// SIMATIC STEP 7 (V5.x) project evaluacion1
// CPU: CPU317-2
// station: Hardware
// station: SIMATIC 300(1)
// station: P_ADR_BUS
// program: S7 Program(1)

SYMBOL_TABLE
"Ejercicio1"	FB 1	FB 1
"Ejercicio 2"	FB 2	FB 2
"Ejercicio3"	FB 3	FB 3
"Ejercicio 4"	FB 4	FB 4
"Ejercicio 5"	FB 5	FB 5
"Ejercicio 6"	FB 6	FB 6
"Ejercicio C1"	FB 7	FB 7
"Ejercicio C2"	FB 8	FB 8
"Ejercicio 3-5"	FB 9	FB 9
"Ejercicio 3-6"	FB 10	FB 10
"Ejercicio 3-7"	FB 11	FB 11
"Ejercicio 6-1"	FB 12	FB 12
"Ejercicio 6-2"	FB 13	FB 13
"Ejercicio 6-3"	FB 14	FB 14
"Paro de emergencia"	FB 99	FB 99
"CYCL_EXC"	OB 1	OB 1	// Cycle Execution
END_SYMBOL_TABLE

FUNCTION_BLOCK "Ejercicio1"	// FB 1
TITLE = Ejercicio 1
VERSION : 0.1
VAR_INPUT
  C_CONTINUO : BOOL ;
  C_UNICO : BOOL ;
  PARO : BOOL ;
  DET_PIEZA : BOOL ;
  A0 : BOOL ;
  A1 : BOOL ;
  B0 : BOOL ;
  B1 : BOOL ;
  C0 : BOOL ;
  C1 : BOOL ;
END_VAR
VAR_OUTPUT
  Y1 : BOOL ;
  Y2 : BOOL ;
  Y3 : BOOL ;
  Y4 : BOOL ;
  Y5 : BOOL ;
  Y6 : BOOL ;
END_VAR
VAR
  K_UNI : BOOL ;
  K_CON : BOOL ;
  K0 : BOOL ;
  K1 : BOOL ;
  K2 : BOOL ;
  K3 : BOOL ;
  K4 : BOOL ;
  K5 : BOOL ;
  K6 : BOOL ;
END_VAR
BEGIN
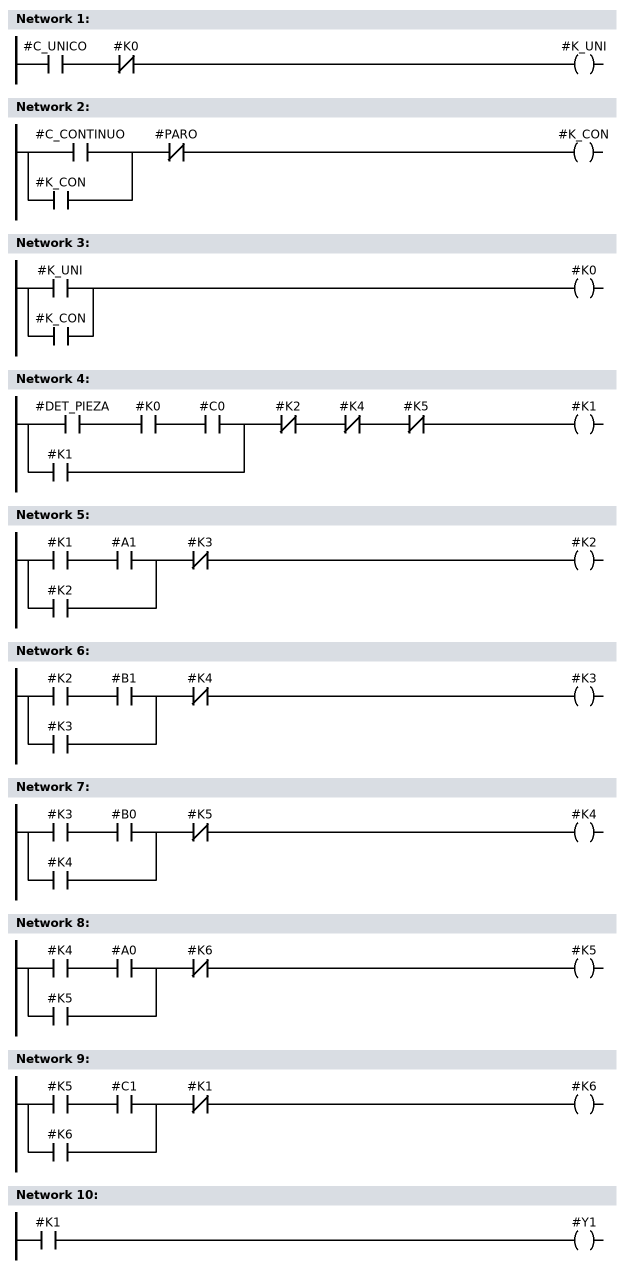
NETWORK
TITLE =
      A     #C_UNICO;
      AN    #K0;
      =     #K_UNI;
NETWORK
TITLE =
      A(;
      O     #C_CONTINUO;
      O     #K_CON;
      );
      AN    #PARO;
      =     #K_CON;
NETWORK
TITLE =
      O     #K_UNI;
      O     #K_CON;
      =     #K0;
NETWORK
TITLE =
      A(;
      A     #DET_PIEZA;
      A     #K0;
      A     #C0;
      O     #K1;
      );
      AN    #K2;
      AN    #K4;
      AN    #K5;
      =     #K1;
NETWORK
TITLE =
      A(;
      A     #K1;
      A     #A1;
      O     #K2;
      );
      AN    #K3;
      =     #K2;
NETWORK
TITLE =
      A(;
      A     #K2;
      A     #B1;
      O     #K3;
      );
      AN    #K4;
      =     #K3;
NETWORK
TITLE =
      A(;
      A     #K3;
      A     #B0;
      O     #K4;
      );
      AN    #K5;
      =     #K4;
NETWORK
TITLE =
      A(;
      A     #K4;
      A     #A0;
      O     #K5;
      );
      AN    #K6;
      =     #K5;
NETWORK
TITLE =
      A(;
      A     #K5;
      A     #C1;
      O     #K6;
      );
      AN    #K1;
      =     #K6;
NETWORK
TITLE =
      A     #K1;
      =     #Y1;
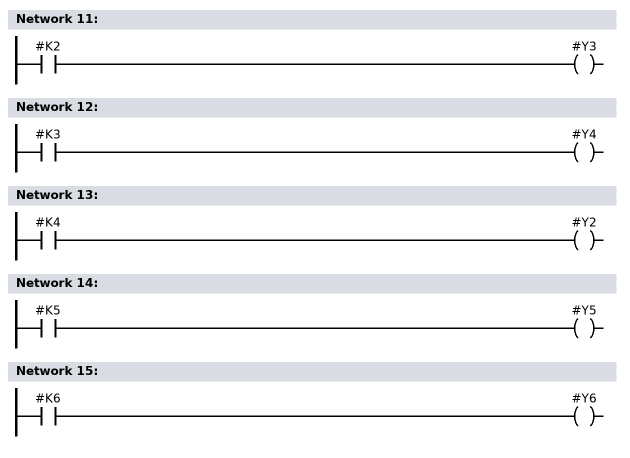
NETWORK
TITLE =
      A     #K2;
      =     #Y3;
NETWORK
TITLE =
      A     #K3;
      =     #Y4;
NETWORK
TITLE =
      A     #K4;
      =     #Y2;
NETWORK
TITLE =
      A     #K5;
      =     #Y5;
NETWORK
TITLE =
      A     #K6;
      =     #Y6;
END_FUNCTION_BLOCK

FUNCTION_BLOCK "Ejercicio 2"	// FB 2
TITLE = Ejercicio 2
VERSION : 0.1
VAR_INPUT
  C_UNICO : BOOL ;
  A0 : BOOL ;
  A1 : BOOL ;
  B0 : BOOL ;
  B1 : BOOL ;
  C0 : BOOL ;
  C1 : BOOL ;
END_VAR
VAR_OUTPUT
  Y1 : BOOL ;
  Y2 : BOOL ;
  Y3 : BOOL ;
  Y4 : BOOL ;
  Y5 : BOOL ;
  Y6 : BOOL ;
END_VAR
VAR
  K_UNI : BOOL ;
  K0 : BOOL ;
  K1 : BOOL ;
  K2 : BOOL ;
  K3 : BOOL ;
  K4 : BOOL ;
  K5 : BOOL ;
  K6 : BOOL ;
END_VAR
BEGIN
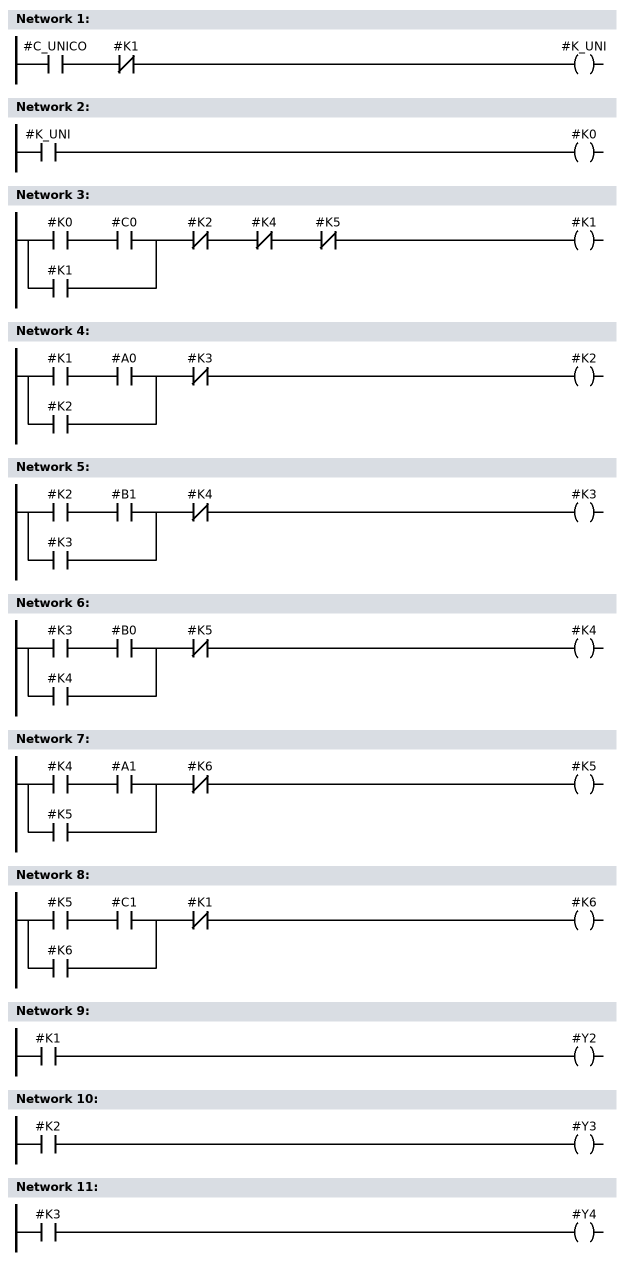
NETWORK
TITLE =
      A     #C_UNICO;
      AN    #K1;
      =     #K_UNI;
NETWORK
TITLE =
      A     #K_UNI;
      =     #K0;
NETWORK
TITLE =
      A(;
      A     #K0;
      A     #C0;
      O     #K1;
      );
      AN    #K2;
      AN    #K4;
      AN    #K5;
      =     #K1;
NETWORK
TITLE =
      A(;
      A     #K1;
      A     #A0;
      O     #K2;
      );
      AN    #K3;
      =     #K2;
NETWORK
TITLE =
      A(;
      A     #K2;
      A     #B1;
      O     #K3;
      );
      AN    #K4;
      =     #K3;
NETWORK
TITLE =
      A(;
      A     #K3;
      A     #B0;
      O     #K4;
      );
      AN    #K5;
      =     #K4;
NETWORK
TITLE =
      A(;
      A     #K4;
      A     #A1;
      O     #K5;
      );
      AN    #K6;
      =     #K5;
NETWORK
TITLE =
      A(;
      A     #K5;
      A     #C1;
      O     #K6;
      );
      AN    #K1;
      =     #K6;
NETWORK
TITLE =
      A     #K1;
      =     #Y2;
NETWORK
TITLE =
      A     #K2;
      =     #Y3;
NETWORK
TITLE =
      A     #K3;
      =     #Y4;
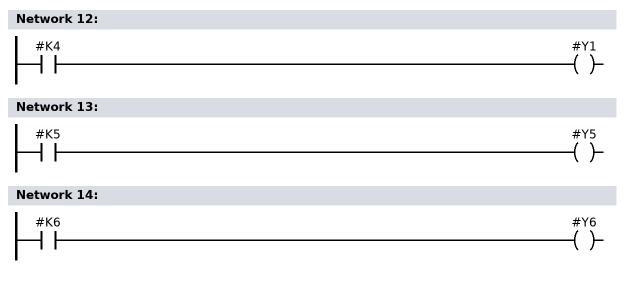
NETWORK
TITLE =
      A     #K4;
      =     #Y1;
NETWORK
TITLE =
      A     #K5;
      =     #Y5;
NETWORK
TITLE =
      A     #K6;
      =     #Y6;
END_FUNCTION_BLOCK

FUNCTION_BLOCK "Ejercicio3"	// FB 3
VERSION : 0.1
VAR_INPUT
  C_UNICO : BOOL ;
  A0 : BOOL ;
  A1 : BOOL ;
  B0 : BOOL ;
  B1 : BOOL ;
  C0 : BOOL ;
  C1 : BOOL ;
END_VAR
VAR_OUTPUT
  Y1 : BOOL ;
  Y2 : BOOL ;
  Y3 : BOOL ;
  Y4 : BOOL ;
  Y5 : BOOL ;
  Y6 : BOOL ;
END_VAR
VAR
  K0 : BOOL ;
  K1 : BOOL ;
  K2 : BOOL ;
  K3 : BOOL ;
  K4 : BOOL ;
  K5 : BOOL ;
  K6 : BOOL ;
  K_UNI : BOOL ;
END_VAR
BEGIN
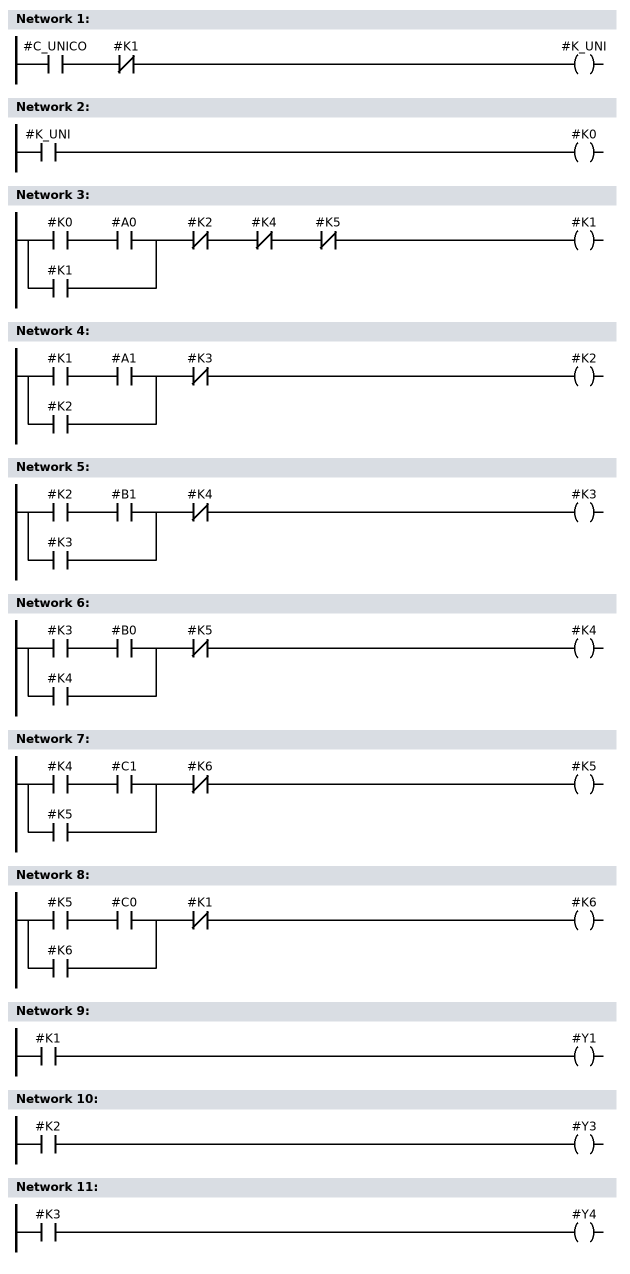
NETWORK
TITLE =
      A     #C_UNICO;
      AN    #K1;
      =     #K_UNI;
NETWORK
TITLE =
      A     #K_UNI;
      =     #K0;
NETWORK
TITLE =
      A(;
      A     #K0;
      A     #A0;
      O     #K1;
      );
      AN    #K2;
      AN    #K4;
      AN    #K5;
      =     #K1;
NETWORK
TITLE =
      A(;
      A     #K1;
      A     #A1;
      O     #K2;
      );
      AN    #K3;
      =     #K2;
NETWORK
TITLE =
      A(;
      A     #K2;
      A     #B1;
      O     #K3;
      );
      AN    #K4;
      =     #K3;
NETWORK
TITLE =
      A(;
      A     #K3;
      A     #B0;
      O     #K4;
      );
      AN    #K5;
      =     #K4;
NETWORK
TITLE =
      A(;
      A     #K4;
      A     #C1;
      O     #K5;
      );
      AN    #K6;
      =     #K5;
NETWORK
TITLE =
      A(;
      A     #K5;
      A     #C0;
      O     #K6;
      );
      AN    #K1;
      =     #K6;
NETWORK
TITLE =
      A     #K1;
      =     #Y1;
NETWORK
TITLE =
      A     #K2;
      =     #Y3;
NETWORK
TITLE =
      A     #K3;
      =     #Y4;
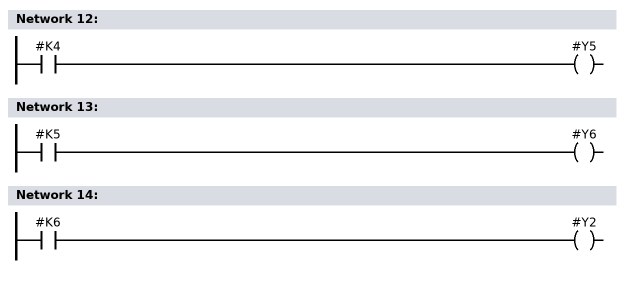
NETWORK
TITLE =
      A     #K4;
      =     #Y5;
NETWORK
TITLE =
      A     #K5;
      =     #Y6;
NETWORK
TITLE =
      A     #K6;
      =     #Y2;
END_FUNCTION_BLOCK

FUNCTION_BLOCK "Ejercicio 4"	// FB 4
VERSION : 0.1
VAR_INPUT
  C_UNICO : BOOL ;
  C_CONTINUO : BOOL ;
  A0 : BOOL ;
  A1 : BOOL ;
  B0 : BOOL ;
  B1 : BOOL ;
  C0 : BOOL ;
  C1 : BOOL ;
  D0 : BOOL ;
  D1 : BOOL ;
  PARO : BOOL ;
END_VAR
VAR_OUTPUT
  Y1 : BOOL ;
  Y2 : BOOL ;
  Y3 : BOOL ;
  Y4 : BOOL ;
  Y5 : BOOL ;
  Y6 : BOOL ;
  Y7 : BOOL ;
  Y8 : BOOL ;
END_VAR
VAR
  K_UNI : BOOL ;
  K_CON : BOOL ;
  K0 : BOOL ;
  K1 : BOOL ;
  K2 : BOOL ;
  K3 : BOOL ;
  K4 : BOOL ;
  K5 : BOOL ;
  K6 : BOOL ;
  K7 : BOOL ;
  K8 : BOOL ;
END_VAR
BEGIN
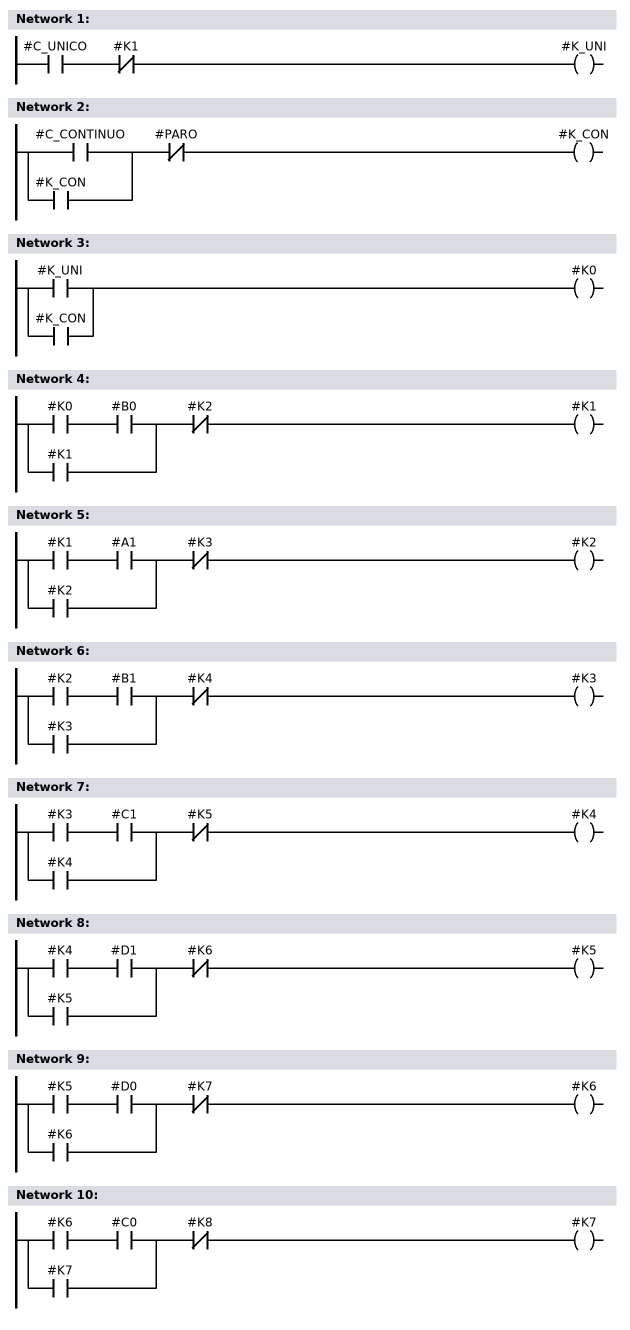
NETWORK
TITLE =
      A     #C_UNICO;
      AN    #K1;
      =     #K_UNI;
NETWORK
TITLE =
      A(;
      O     #C_CONTINUO;
      O     #K_CON;
      );
      AN    #PARO;
      =     #K_CON;
NETWORK
TITLE =
      O     #K_UNI;
      O     #K_CON;
      =     #K0;
NETWORK
TITLE =
      A(;
      A     #K0;
      A     #B0;
      O     #K1;
      );
      AN    #K2;
      =     #K1;
NETWORK
TITLE =
      A(;
      A     #K1;
      A     #A1;
      O     #K2;
      );
      AN    #K3;
      =     #K2;
NETWORK
TITLE =
      A(;
      A     #K2;
      A     #B1;
      O     #K3;
      );
      AN    #K4;
      =     #K3;
NETWORK
TITLE =
      A(;
      A     #K3;
      A     #C1;
      O     #K4;
      );
      AN    #K5;
      =     #K4;
NETWORK
TITLE =
      A(;
      A     #K4;
      A     #D1;
      O     #K5;
      );
      AN    #K6;
      =     #K5;
NETWORK
TITLE =
      A(;
      A     #K5;
      A     #D0;
      O     #K6;
      );
      AN    #K7;
      =     #K6;
NETWORK
TITLE =
      A(;
      A     #K6;
      A     #C0;
      O     #K7;
      );
      AN    #K8;
      =     #K7;
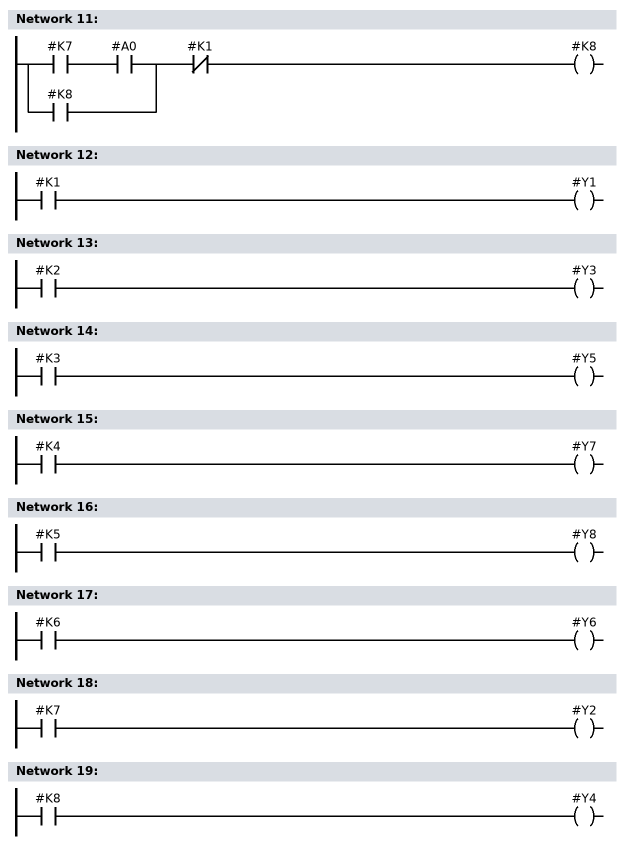
NETWORK
TITLE =
      A(;
      A     #K7;
      A     #A0;
      O     #K8;
      );
      AN    #K1;
      =     #K8;
NETWORK
TITLE =
      A     #K1;
      =     #Y1;
NETWORK
TITLE =
      A     #K2;
      =     #Y3;
NETWORK
TITLE =
      A     #K3;
      =     #Y5;
NETWORK
TITLE =
      A     #K4;
      =     #Y7;
NETWORK
TITLE =
      A     #K5;
      =     #Y8;
NETWORK
TITLE =
      A     #K6;
      =     #Y6;
NETWORK
TITLE =
      A     #K7;
      =     #Y2;
NETWORK
TITLE =
      A     #K8;
      =     #Y4;
END_FUNCTION_BLOCK

FUNCTION_BLOCK "Ejercicio 5"	// FB 5
VERSION : 0.1
VAR_INPUT
  C_UNICO : BOOL ;
  A0 : BOOL ;
  A1 : BOOL ;
  B0 : BOOL ;
  B1 : BOOL ;
  C0 : BOOL ;
  C1 : BOOL ;
END_VAR
VAR_OUTPUT
  Y1 : BOOL ;
  Y2 : BOOL ;
  Y3 : BOOL ;
  Y4 : BOOL ;
  Y5 : BOOL ;
  Y6 : BOOL ;
END_VAR
VAR
  K_UNI : BOOL ;
  K0 : BOOL ;
  K1 : BOOL ;
  K2 : BOOL ;
  K3 : BOOL ;
  K4 : BOOL ;
  K5 : BOOL ;
  K6 : BOOL ;
  K7 : BOOL ;
  K8 : BOOL ;
  K9 : BOOL ;
  K10 : BOOL ;
END_VAR
BEGIN
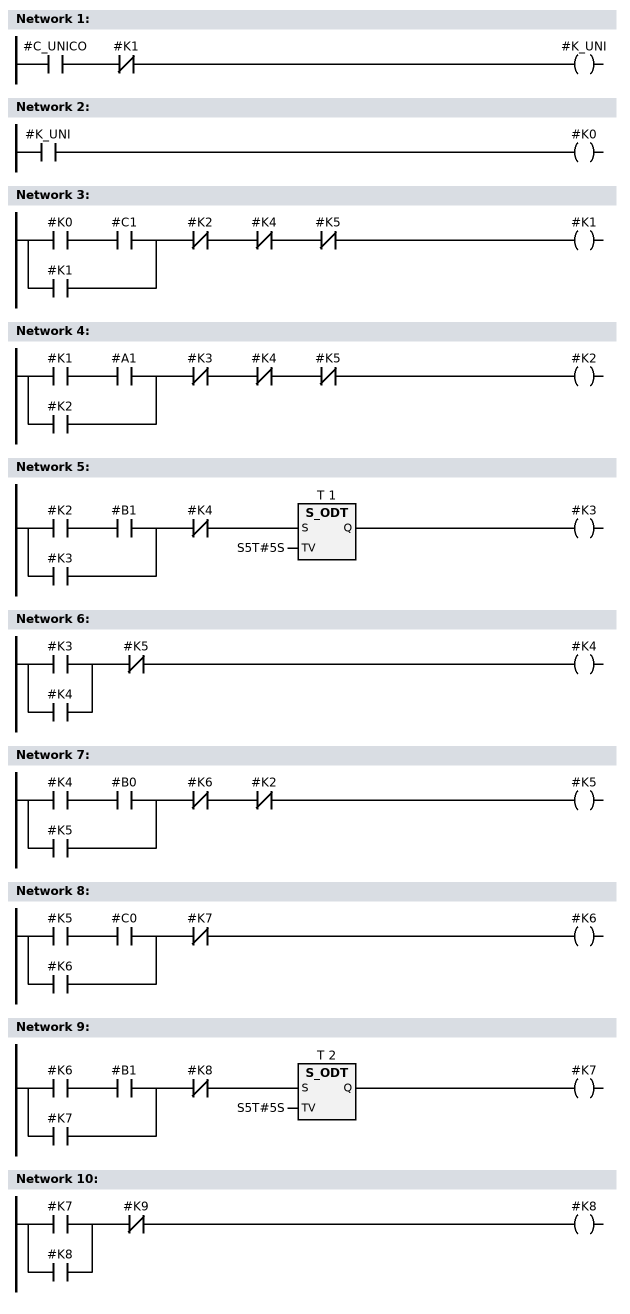
NETWORK
TITLE =
      A     #C_UNICO;
      AN    #K1;
      =     #K_UNI;
NETWORK
TITLE =
      A     #K_UNI;
      =     #K0;
NETWORK
TITLE =
      A(;
      A     #K0;
      A     #C1;
      O     #K1;
      );
      AN    #K2;
      AN    #K4;
      AN    #K5;
      =     #K1;
NETWORK
TITLE =
      A(;
      A     #K1;
      A     #A1;
      O     #K2;
      );
      AN    #K3;
      AN    #K4;
      AN    #K5;
      =     #K2;
NETWORK
TITLE =
      A(;
      A     #K2;
      A     #B1;
      O     #K3;
      );
      AN    #K4;
      L     S5T#5S;
      SD    T 1;
      NOP   0;
      NOP   0;
      NOP   0;
      A     T 1;
      =     #K3;
NETWORK
TITLE =
      A(;
      O     #K3;
      O     #K4;
      );
      AN    #K5;
      =     #K4;
NETWORK
TITLE =
      A(;
      A     #K4;
      A     #B0;
      O     #K5;
      );
      AN    #K6;
      AN    #K2;
      =     #K5;
NETWORK
TITLE =
      A(;
      A     #K5;
      A     #C0;
      O     #K6;
      );
      AN    #K7;
      =     #K6;
NETWORK
TITLE =
      A(;
      A     #K6;
      A     #B1;
      O     #K7;
      );
      AN    #K8;
      L     S5T#5S;
      SD    T 2;
      NOP   0;
      NOP   0;
      NOP   0;
      A     T 2;
      =     #K7;
NETWORK
TITLE =
      A(;
      O     #K7;
      O     #K8;
      );
      AN    #K9;
      =     #K8;
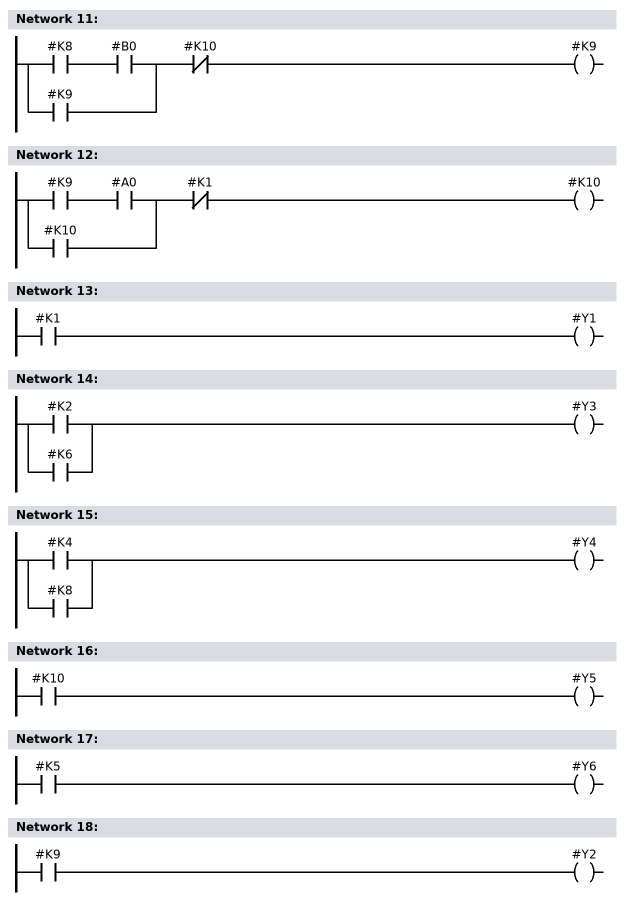
NETWORK
TITLE =
      A(;
      A     #K8;
      A     #B0;
      O     #K9;
      );
      AN    #K10;
      =     #K9;
NETWORK
TITLE =
      A(;
      A     #K9;
      A     #A0;
      O     #K10;
      );
      AN    #K1;
      =     #K10;
NETWORK
TITLE =
      A     #K1;
      =     #Y1;
NETWORK
TITLE =
      O     #K2;
      O     #K6;
      =     #Y3;
NETWORK
TITLE =
      O     #K4;
      O     #K8;
      =     #Y4;
NETWORK
TITLE =
      A     #K10;
      =     #Y5;
NETWORK
TITLE =
      A     #K5;
      =     #Y6;
NETWORK
TITLE =
      A     #K9;
      =     #Y2;
END_FUNCTION_BLOCK

FUNCTION_BLOCK "Ejercicio 6"	// FB 6
VERSION : 0.1
VAR_INPUT
  C_UNICO : BOOL ;
  C_CONTINUO : BOOL ;
  PARO : BOOL ;
  A0 : BOOL ;
  A1 : BOOL ;
  B0 : BOOL ;
  B1 : BOOL ;
  C0 : BOOL ;
  C1 : BOOL ;
  D0 : BOOL ;
  D1 : BOOL ;
END_VAR
VAR_OUTPUT
  Y1 : BOOL ;
  Y2 : BOOL ;
  Y3 : BOOL ;
  Y4 : BOOL ;
  Y5 : BOOL ;
  Y6 : BOOL ;
  Y7 : BOOL ;
  Y8 : BOOL ;
END_VAR
VAR
  K0 : BOOL ;
  K1 : BOOL ;
  K2 : BOOL ;
  K3 : BOOL ;
  K4 : BOOL ;
  K5 : BOOL ;
  K6 : BOOL ;
  K7 : BOOL ;
  K8 : BOOL ;
  KA : BOOL ;
  KB : BOOL ;
END_VAR
BEGIN
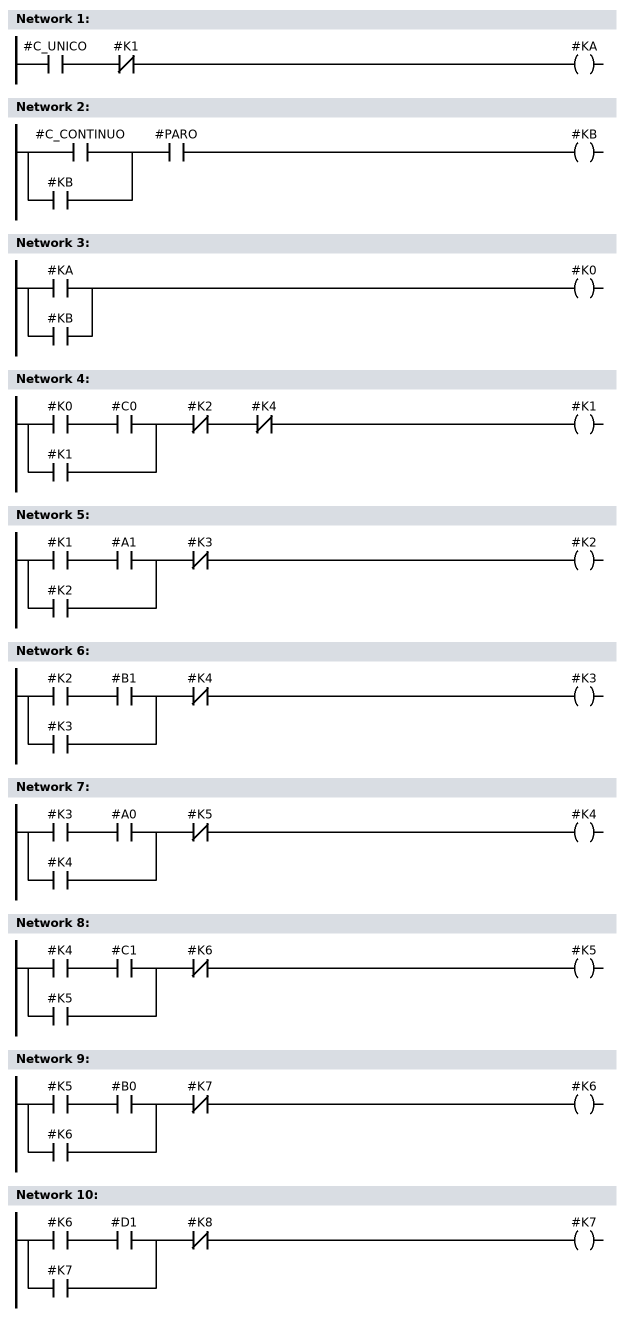
NETWORK
TITLE =
      A     #C_UNICO;
      AN    #K1;
      =     #KA;
NETWORK
TITLE =
      A(;
      O     #C_CONTINUO;
      O     #KB;
      );
      A     #PARO;
      =     #KB;
NETWORK
TITLE =
      O     #KA;
      O     #KB;
      =     #K0;
NETWORK
TITLE =
      A(;
      A     #K0;
      A     #C0;
      O     #K1;
      );
      AN    #K2;
      AN    #K4;
      =     #K1;
NETWORK
TITLE =
      A(;
      A     #K1;
      A     #A1;
      O     #K2;
      );
      AN    #K3;
      =     #K2;
NETWORK
TITLE =
      A(;
      A     #K2;
      A     #B1;
      O     #K3;
      );
      AN    #K4;
      =     #K3;
NETWORK
TITLE =
      A(;
      A     #K3;
      A     #A0;
      O     #K4;
      );
      AN    #K5;
      =     #K4;
NETWORK
TITLE =
      A(;
      A     #K4;
      A     #C1;
      O     #K5;
      );
      AN    #K6;
      =     #K5;
NETWORK
TITLE =
      A(;
      A     #K5;
      A     #B0;
      O     #K6;
      );
      AN    #K7;
      =     #K6;
NETWORK
TITLE =
      A(;
      A     #K6;
      A     #D1;
      O     #K7;
      );
      AN    #K8;
      =     #K7;
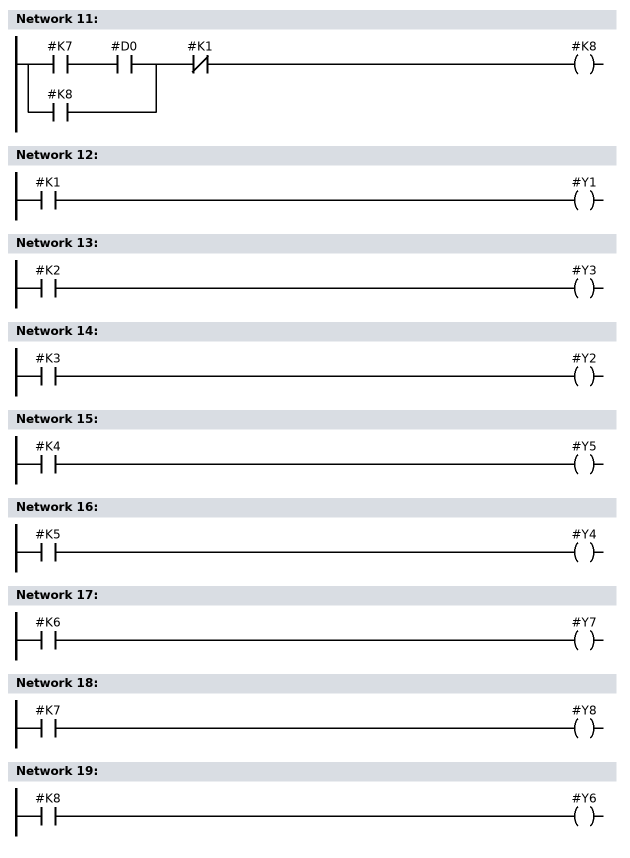
NETWORK
TITLE =
      A(;
      A     #K7;
      A     #D0;
      O     #K8;
      );
      AN    #K1;
      =     #K8;
NETWORK
TITLE =
      A     #K1;
      =     #Y1;
NETWORK
TITLE =
      A     #K2;
      =     #Y3;
NETWORK
TITLE =
      A     #K3;
      =     #Y2;
NETWORK
TITLE =
      A     #K4;
      =     #Y5;
NETWORK
TITLE =
      A     #K5;
      =     #Y4;
NETWORK
TITLE =
      A     #K6;
      =     #Y7;
NETWORK
TITLE =
      A     #K7;
      =     #Y8;
NETWORK
TITLE =
      A     #K8;
      =     #Y6;
END_FUNCTION_BLOCK

FUNCTION_BLOCK "Ejercicio C1"	// FB 7
VERSION : 0.1
VAR_INPUT
  C_UNICO : BOOL ;
  C_CONTINUO : BOOL ;
  PARO : BOOL ;
  C_BROCA : BOOL ;
  A0 : BOOL ;
  A1 : BOOL ;
  B0 : BOOL ;
  B1 : BOOL ;
  C0 : BOOL ;
  C1 : BOOL ;
END_VAR
VAR_OUTPUT
  Y1 : BOOL ;
  Y2 : BOOL ;
  Y3 : BOOL ;
  Y4 : BOOL ;
  Y5 : BOOL ;
  Y6 : BOOL ;
END_VAR
VAR
  K0 : BOOL ;
  K1 : BOOL ;
  K2 : BOOL ;
  K3 : BOOL ;
  K4 : BOOL ;
  K5 : BOOL ;
  K6 : BOOL ;
  KA : BOOL ;
  KB : BOOL ;
  CNT : BOOL ;
  K7 : BOOL ;
  K8 : BOOL ;
  K9 : BOOL ;
  K10 : BOOL ;
  K11 : BOOL ;
  K12 : BOOL ;
END_VAR
BEGIN
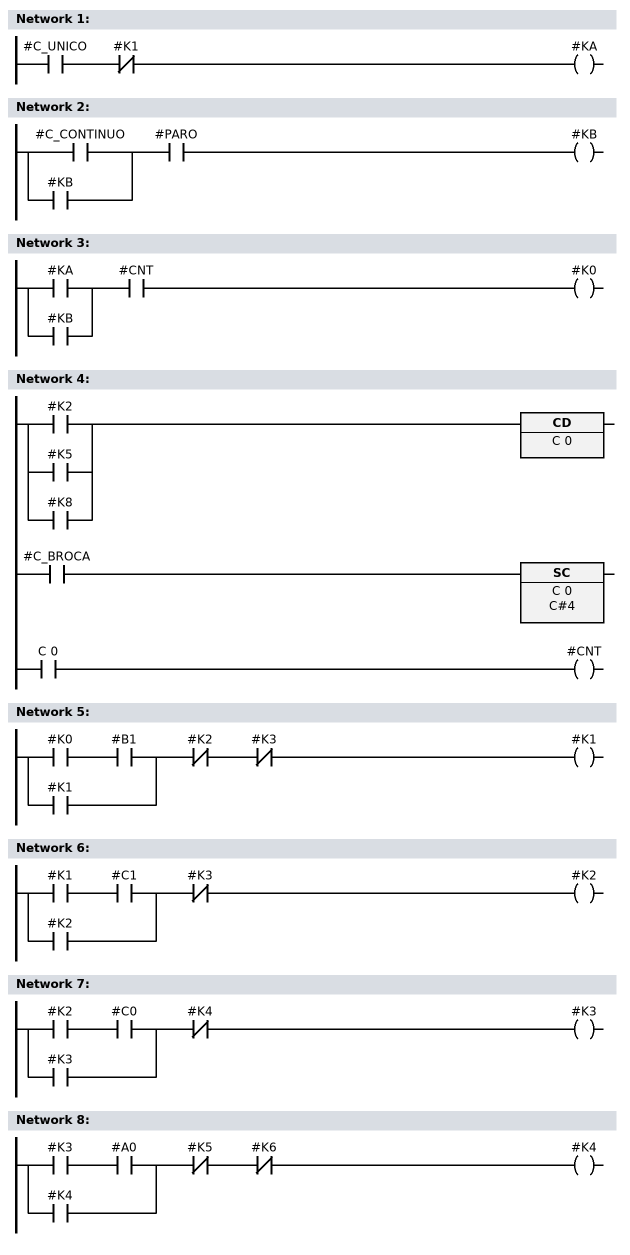
NETWORK
TITLE =
      A     #C_UNICO;
      AN    #K1;
      =     #KA;
NETWORK
TITLE =
      A(;
      O     #C_CONTINUO;
      O     #KB;
      );
      A     #PARO;
      =     #KB;
NETWORK
TITLE =
      A(;
      O     #KA;
      O     #KB;
      );
      A     #CNT;
      =     #K0;
NETWORK
TITLE =
      A(;
      O     #K2;
      O     #K5;
      O     #K8;
      );
      CD    C 0;
      BLD   101;
      A     #C_BROCA;
      L     C#4;
      S     C 0;
      NOP   0;
      NOP   0;
      NOP   0;
      A     C 0;
      =     #CNT;
NETWORK
TITLE =
      A(;
      A     #K0;
      A     #B1;
      O     #K1;
      );
      AN    #K2;
      AN    #K3;
      =     #K1;
NETWORK
TITLE =
      A(;
      A     #K1;
      A     #C1;
      O     #K2;
      );
      AN    #K3;
      =     #K2;
NETWORK
TITLE =
      A(;
      A     #K2;
      A     #C0;
      O     #K3;
      );
      AN    #K4;
      =     #K3;
NETWORK
TITLE =
      A(;
      A     #K3;
      A     #A0;
      O     #K4;
      );
      AN    #K5;
      AN    #K6;
      =     #K4;
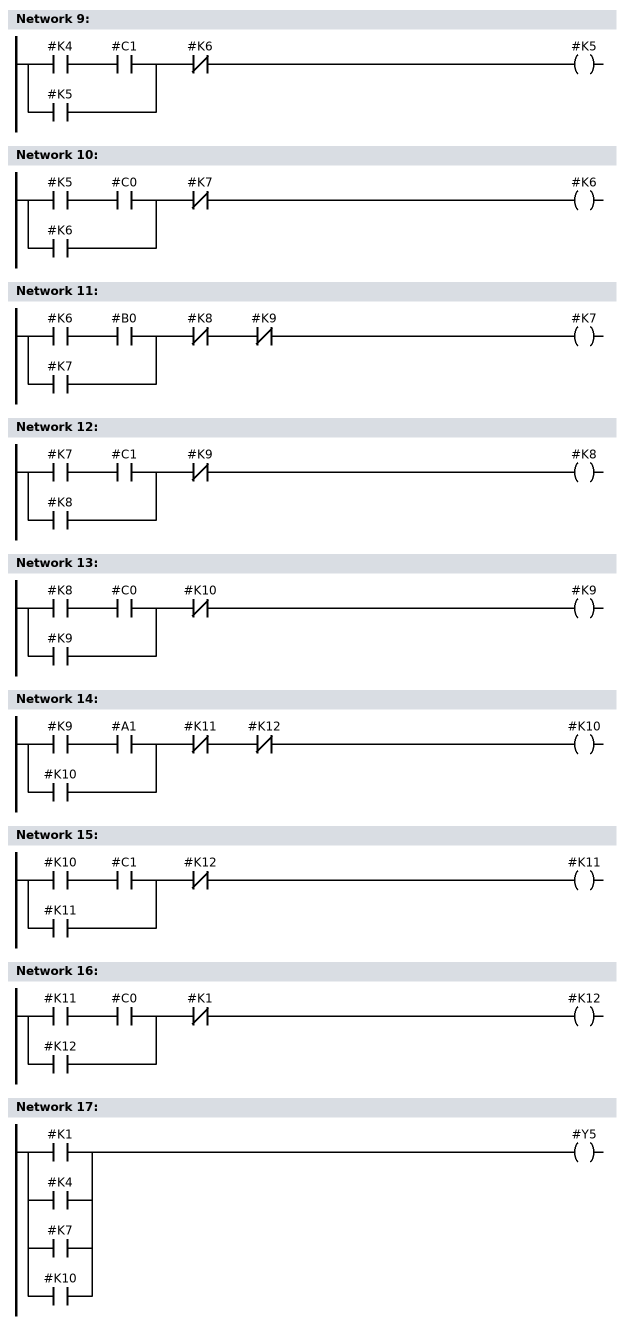
NETWORK
TITLE =
      A(;
      A     #K4;
      A     #C1;
      O     #K5;
      );
      AN    #K6;
      =     #K5;
NETWORK
TITLE =
      A(;
      A     #K5;
      A     #C0;
      O     #K6;
      );
      AN    #K7;
      =     #K6;
NETWORK
TITLE =
      A(;
      A     #K6;
      A     #B0;
      O     #K7;
      );
      AN    #K8;
      AN    #K9;
      =     #K7;
NETWORK
TITLE =
      A(;
      A     #K7;
      A     #C1;
      O     #K8;
      );
      AN    #K9;
      =     #K8;
NETWORK
TITLE =
      A(;
      A     #K8;
      A     #C0;
      O     #K9;
      );
      AN    #K10;
      =     #K9;
NETWORK
TITLE =
      A(;
      A     #K9;
      A     #A1;
      O     #K10;
      );
      AN    #K11;
      AN    #K12;
      =     #K10;
NETWORK
TITLE =
      A(;
      A     #K10;
      A     #C1;
      O     #K11;
      );
      AN    #K12;
      =     #K11;
NETWORK
TITLE =
      A(;
      A     #K11;
      A     #C0;
      O     #K12;
      );
      AN    #K1;
      =     #K12;
NETWORK
TITLE =
      O     #K1;
      O     #K4;
      O     #K7;
      O     #K10;
      =     #Y5;
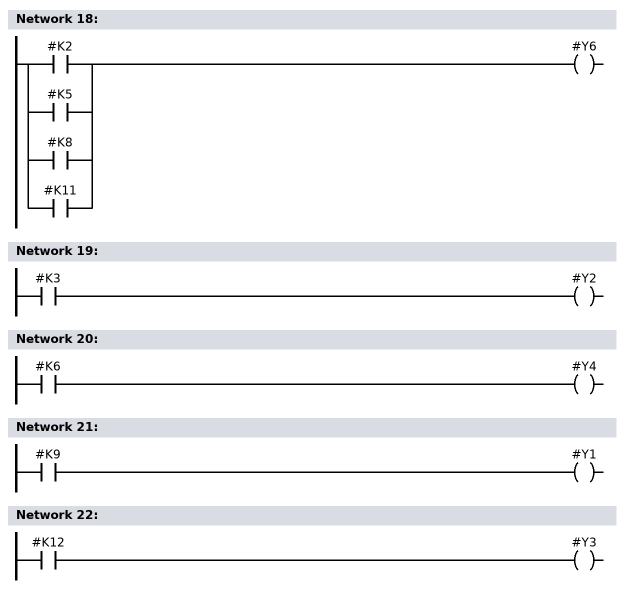
NETWORK
TITLE =
      O     #K2;
      O     #K5;
      O     #K8;
      O     #K11;
      =     #Y6;
NETWORK
TITLE =
      A     #K3;
      =     #Y2;
NETWORK
TITLE =
      A     #K6;
      =     #Y4;
NETWORK
TITLE =
      A     #K9;
      =     #Y1;
NETWORK
TITLE =
      A     #K12;
      =     #Y3;
END_FUNCTION_BLOCK

FUNCTION_BLOCK "Ejercicio C2"	// FB 8
VERSION : 0.1
VAR_INPUT
  C_UNICO : BOOL ;
  C_CONTINUO : BOOL ;
  PARO : BOOL ;
  DET_PIEZA : BOOL ;
  DET_CINTA : BOOL ;
  A0 : BOOL ;
  A1 : BOOL ;
  B0 : BOOL ;
  B1 : BOOL ;
  C0 : BOOL ;
  C1 : BOOL ;
  D0 : BOOL ;
  D1 : BOOL ;
  E0 : BOOL ;
  E1 : BOOL ;
  F0 : BOOL ;
  F1 : BOOL ;
END_VAR
VAR_OUTPUT
  Y1 : BOOL ;
  Y2 : BOOL ;
  Y3 : BOOL ;
  Y4 : BOOL ;
  Y5 : BOOL ;
  Y6 : BOOL ;
  Y7 : BOOL ;
  Y8 : BOOL ;
  Y9 : BOOL ;
  Y10 : BOOL ;
  Y11 : BOOL ;
  Y12 : BOOL ;
END_VAR
VAR
  KA : BOOL ;
  KB : BOOL ;
  K0 : BOOL ;
  K1 : BOOL ;
  K2 : BOOL ;
  K3 : BOOL ;
  K4 : BOOL ;
  K5 : BOOL ;
  K6 : BOOL ;
  K7 : BOOL ;
  K8 : BOOL ;
  K9 : BOOL ;
  K10 : BOOL ;
  K11 : BOOL ;
END_VAR
BEGIN
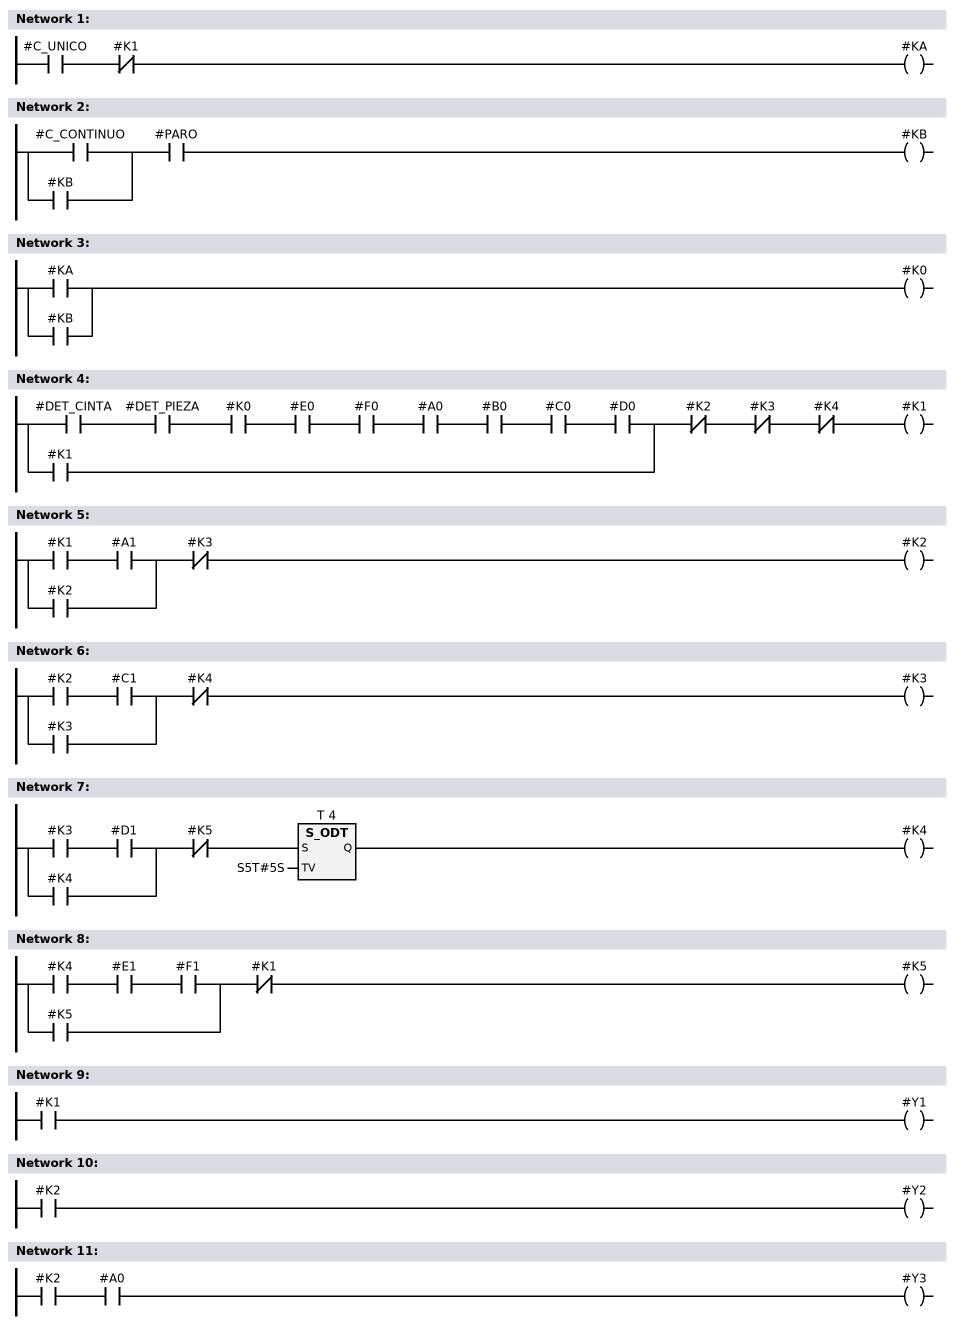
NETWORK
TITLE =
      A     #C_UNICO;
      AN    #K1;
      =     #KA;
NETWORK
TITLE =
      A(;
      O     #C_CONTINUO;
      O     #KB;
      );
      A     #PARO;
      =     #KB;
NETWORK
TITLE =
      O     #KA;
      O     #KB;
      =     #K0;
NETWORK
TITLE =
      A(;
      A     #DET_CINTA;
      A     #DET_PIEZA;
      A     #K0;
      A     #E0;
      A     #F0;
      A     #A0;
      A     #B0;
      A     #C0;
      A     #D0;
      O     #K1;
      );
      AN    #K2;
      AN    #K3;
      AN    #K4;
      =     #K1;
NETWORK
TITLE =
      A(;
      A     #K1;
      A     #A1;
      O     #K2;
      );
      AN    #K3;
      =     #K2;
NETWORK
TITLE =
      A(;
      A     #K2;
      A     #C1;
      O     #K3;
      );
      AN    #K4;
      =     #K3;
NETWORK
TITLE =
      A(;
      A     #K3;
      A     #D1;
      O     #K4;
      );
      AN    #K5;
      L     S5T#5S;
      SD    T 4;
      NOP   0;
      NOP   0;
      NOP   0;
      A     T 4;
      =     #K4;
NETWORK
TITLE =
      A(;
      A     #K4;
      A     #E1;
      A     #F1;
      O     #K5;
      );
      AN    #K1;
      =     #K5;
NETWORK
TITLE =
      A     #K1;
      =     #Y1;
NETWORK
TITLE =
      A     #K2;
      =     #Y2;
NETWORK
TITLE =
      A     #K2;
      A     #A0;
      =     #Y3;
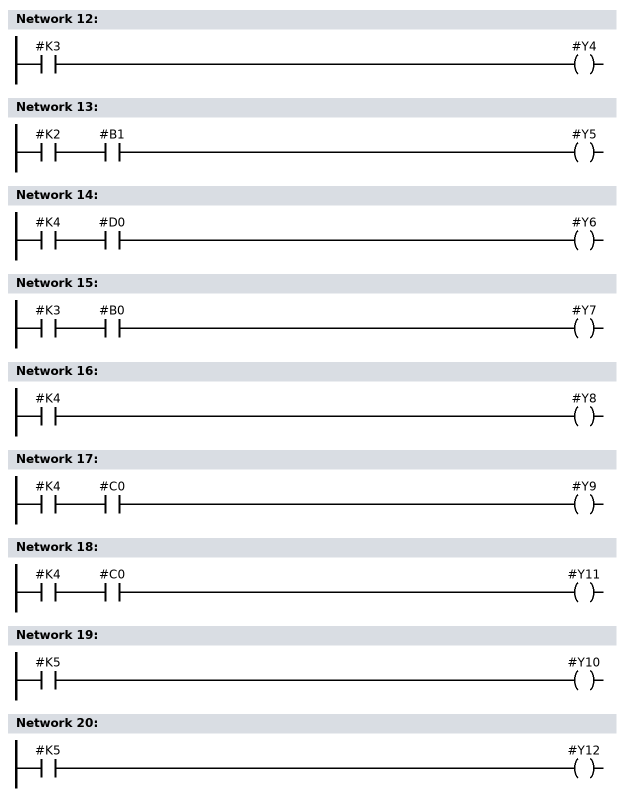
NETWORK
TITLE =
      A     #K3;
      =     #Y4;
NETWORK
TITLE =
      A     #K2;
      A     #B1;
      =     #Y5;
NETWORK
TITLE =
      A     #K4;
      A     #D0;
      =     #Y6;
NETWORK
TITLE =
      A     #K3;
      A     #B0;
      =     #Y7;
NETWORK
TITLE =
      A     #K4;
      =     #Y8;
NETWORK
TITLE =
      A     #K4;
      A     #C0;
      =     #Y9;
NETWORK
TITLE =
      A     #K4;
      A     #C0;
      =     #Y11;
NETWORK
TITLE =
      A     #K5;
      =     #Y10;
NETWORK
TITLE =
      A     #K5;
      =     #Y12;
END_FUNCTION_BLOCK

FUNCTION_BLOCK "Ejercicio 3-5"	// FB 9
VERSION : 0.1
VAR_INPUT
  C_UNICO : BOOL ;
  A0 : BOOL ;
  A1 : BOOL ;
  B0 : BOOL ;
  B1 : BOOL ;
  C0 : BOOL ;
  C1 : BOOL ;
  D0 : BOOL ;
  D1 : BOOL ;
  HONGO : BOOL ;
  RESET : BOOL ;
END_VAR
VAR_OUTPUT
  Y1 : BOOL ;
  Y2 : BOOL ;
  Y3 : BOOL ;
  Y4 : BOOL ;
  Y5 : BOOL ;
  Y6 : BOOL ;
  Y7 : BOOL ;
  Y8 : BOOL ;
END_VAR
VAR
  KA : BOOL ;
  K0 : BOOL ;
  K1 : BOOL ;
  K2 : BOOL ;
  K3 : BOOL ;
  K4 : BOOL ;
  K5 : BOOL ;
  K6 : BOOL ;
  K7 : BOOL ;
  K8 : BOOL ;
  K9 : BOOL ;
  K10 : BOOL ;
  K_PEM : BOOL ;
END_VAR
BEGIN
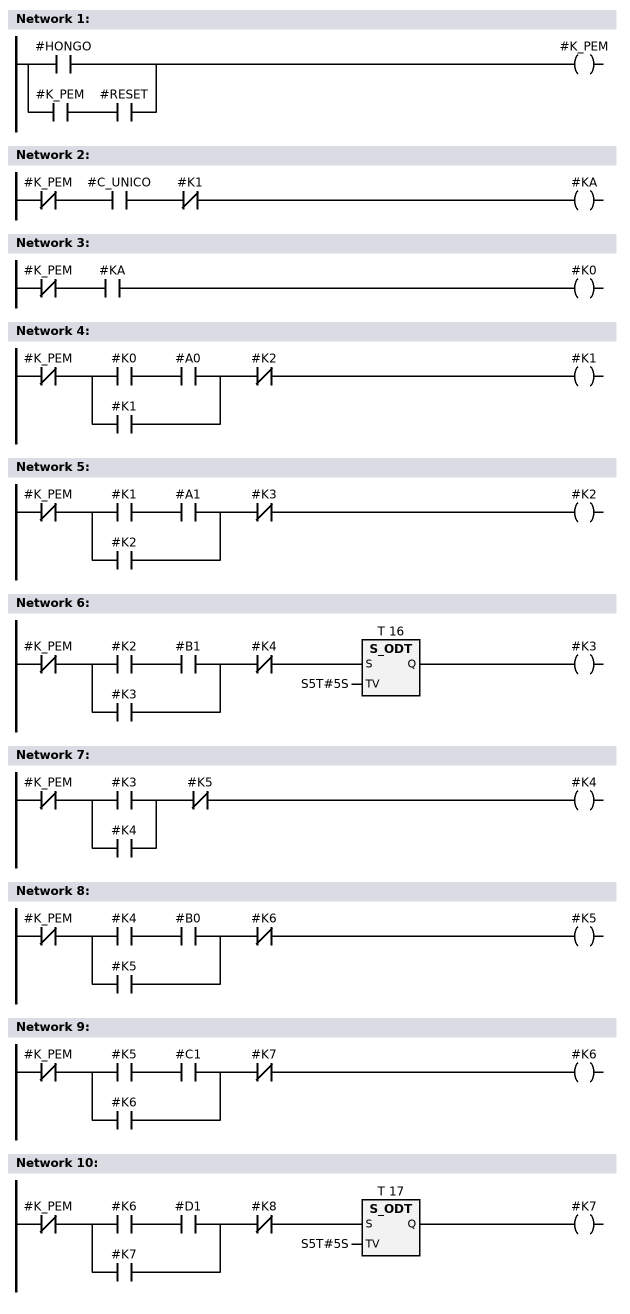
NETWORK
TITLE =
      O     #HONGO;
      O;
      A     #K_PEM;
      A     #RESET;
      =     #K_PEM;
NETWORK
TITLE =
      AN    #K_PEM;
      A     #C_UNICO;
      AN    #K1;
      =     #KA;
NETWORK
TITLE =
      AN    #K_PEM;
      A     #KA;
      =     #K0;
NETWORK
TITLE =
      AN    #K_PEM;
      A(;
      A     #K0;
      A     #A0;
      O     #K1;
      );
      AN    #K2;
      =     #K1;
NETWORK
TITLE =
      AN    #K_PEM;
      A(;
      A     #K1;
      A     #A1;
      O     #K2;
      );
      AN    #K3;
      =     #K2;
NETWORK
TITLE =
      AN    #K_PEM;
      A(;
      A     #K2;
      A     #B1;
      O     #K3;
      );
      AN    #K4;
      L     S5T#5S;
      SD    T 16;
      NOP   0;
      NOP   0;
      NOP   0;
      A     T 16;
      =     #K3;
NETWORK
TITLE =
      AN    #K_PEM;
      A(;
      O     #K3;
      O     #K4;
      );
      AN    #K5;
      =     #K4;
NETWORK
TITLE =
      AN    #K_PEM;
      A(;
      A     #K4;
      A     #B0;
      O     #K5;
      );
      AN    #K6;
      =     #K5;
NETWORK
TITLE =
      AN    #K_PEM;
      A(;
      A     #K5;
      A     #C1;
      O     #K6;
      );
      AN    #K7;
      =     #K6;
NETWORK
TITLE =
      AN    #K_PEM;
      A(;
      A     #K6;
      A     #D1;
      O     #K7;
      );
      AN    #K8;
      L     S5T#5S;
      SD    T 17;
      NOP   0;
      NOP   0;
      NOP   0;
      A     T 17;
      =     #K7;
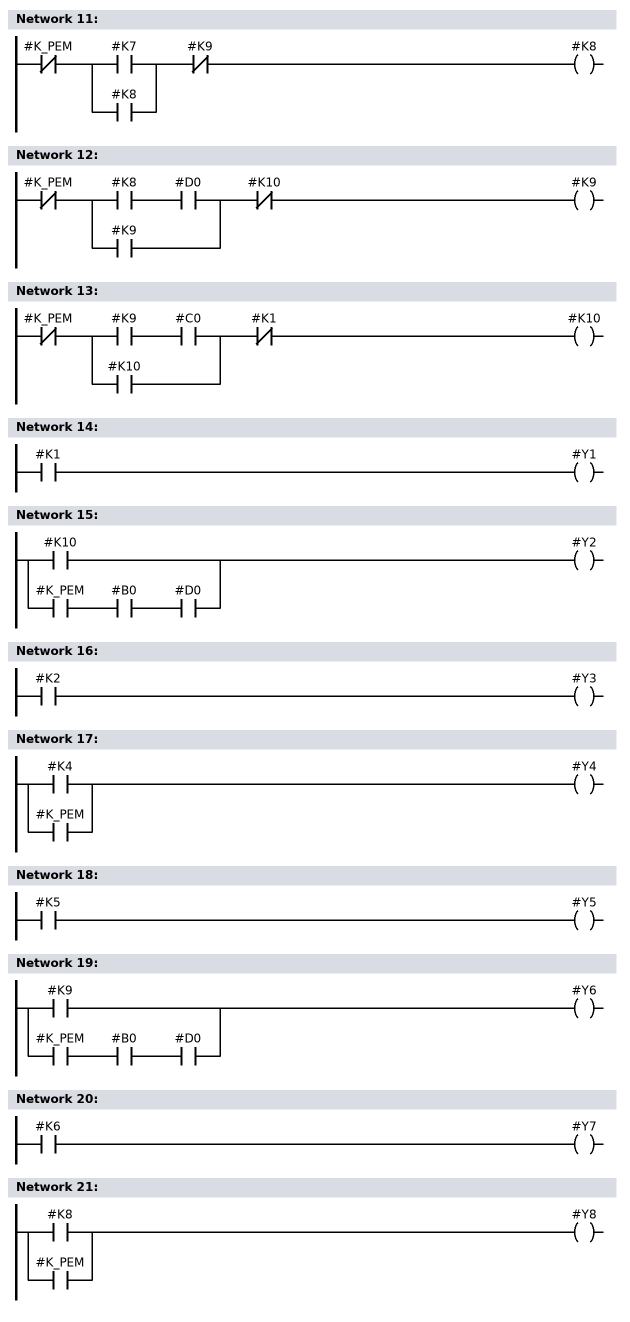
NETWORK
TITLE =
      AN    #K_PEM;
      A(;
      O     #K7;
      O     #K8;
      );
      AN    #K9;
      =     #K8;
NETWORK
TITLE =
      AN    #K_PEM;
      A(;
      A     #K8;
      A     #D0;
      O     #K9;
      );
      AN    #K10;
      =     #K9;
NETWORK
TITLE =
      AN    #K_PEM;
      A(;
      A     #K9;
      A     #C0;
      O     #K10;
      );
      AN    #K1;
      =     #K10;
NETWORK
TITLE =
      A     #K1;
      =     #Y1;
NETWORK
TITLE =
      O     #K10;
      O;
      A     #K_PEM;
      A     #B0;
      A     #D0;
      =     #Y2;
NETWORK
TITLE =
      A     #K2;
      =     #Y3;
NETWORK
TITLE =
      O     #K4;
      O     #K_PEM;
      =     #Y4;
NETWORK
TITLE =
      A     #K5;
      =     #Y5;
NETWORK
TITLE =
      O     #K9;
      O;
      A     #K_PEM;
      A     #B0;
      A     #D0;
      =     #Y6;
NETWORK
TITLE =
      A     #K6;
      =     #Y7;
NETWORK
TITLE =
      O     #K8;
      O     #K_PEM;
      =     #Y8;
END_FUNCTION_BLOCK

FUNCTION_BLOCK "Ejercicio 3-6"	// FB 10
VERSION : 0.1
VAR_INPUT
  C_UNICO : BOOL ;
  C_CONTINUO : BOOL ;
  PARO : BOOL ;
  DET_PIEZA : BOOL ;
  A0 : BOOL ;
  A1 : BOOL ;
  B0 : BOOL ;
  B1 : BOOL ;
  C0 : BOOL ;
  C1 : BOOL ;
  D0 : BOOL ;
  D1 : BOOL ;
END_VAR
VAR_OUTPUT
  Y1 : BOOL ;
  Y2 : BOOL ;
  Y3 : BOOL ;
  Y4 : BOOL ;
  Y5 : BOOL ;
  Y6 : BOOL ;
  Y7 : BOOL ;
  Y8 : BOOL ;
END_VAR
VAR
  KA : BOOL ;
  KB : BOOL ;
  K0 : BOOL ;
  K1 : BOOL ;
  K2 : BOOL ;
  K3 : BOOL ;
  K4 : BOOL ;
  K5 : BOOL ;
  K6 : BOOL ;
  K7 : BOOL ;
  K8 : BOOL ;
  K9 : BOOL ;
END_VAR
BEGIN
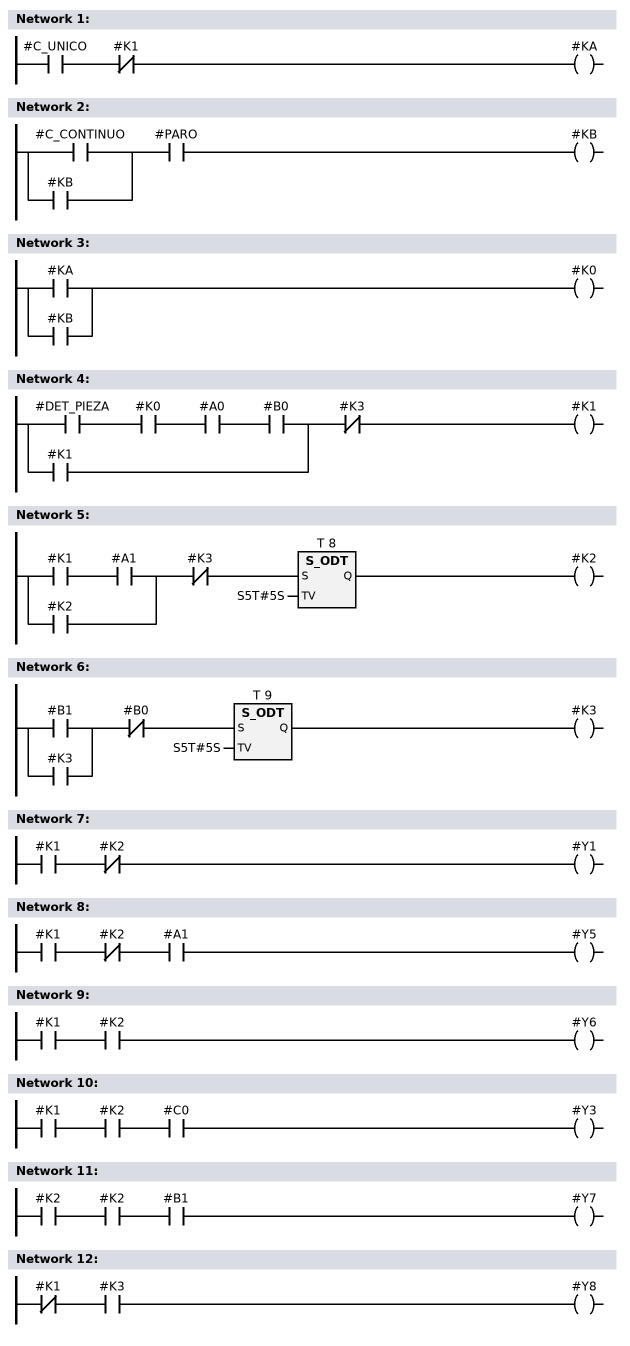
NETWORK
TITLE =
      A     #C_UNICO;
      AN    #K1;
      =     #KA;
NETWORK
TITLE =
      A(;
      O     #C_CONTINUO;
      O     #KB;
      );
      A     #PARO;
      =     #KB;
NETWORK
TITLE =
      O     #KA;
      O     #KB;
      =     #K0;
NETWORK
TITLE =
      A(;
      A     #DET_PIEZA;
      A     #K0;
      A     #A0;
      A     #B0;
      O     #K1;
      );
      AN    #K3;
      =     #K1;
NETWORK
TITLE =
      A(;
      A     #K1;
      A     #A1;
      O     #K2;
      );
      AN    #K3;
      L     S5T#5S;
      SD    T 8;
      NOP   0;
      NOP   0;
      NOP   0;
      A     T 8;
      =     #K2;
NETWORK
TITLE =
      A(;
      O     #B1;
      O     #K3;
      );
      AN    #B0;
      L     S5T#5S;
      SD    T 9;
      NOP   0;
      NOP   0;
      NOP   0;
      A     T 9;
      =     #K3;
NETWORK
TITLE =
      A     #K1;
      AN    #K2;
      =     #Y1;
NETWORK
TITLE =
      A     #K1;
      AN    #K2;
      A     #A1;
      =     #Y5;
NETWORK
TITLE =
      A     #K1;
      A     #K2;
      =     #Y6;
NETWORK
TITLE =
      A     #K1;
      A     #K2;
      A     #C0;
      =     #Y3;
NETWORK
TITLE =
      A     #K2;
      A     #K2;
      A     #B1;
      =     #Y7;
NETWORK
TITLE =
      AN    #K1;
      A     #K3;
      =     #Y8;
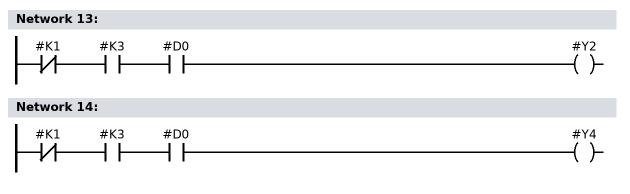
NETWORK
TITLE =
      AN    #K1;
      A     #K3;
      A     #D0;
      =     #Y2;
NETWORK
TITLE =
      AN    #K1;
      A     #K3;
      A     #D0;
      =     #Y4;
END_FUNCTION_BLOCK

FUNCTION_BLOCK "Ejercicio 3-7"	// FB 11
VERSION : 0.1
VAR_INPUT
  C_UNICO : BOOL ;
  C_CONTINUO : BOOL ;
  PARO : BOOL ;
  DET_PIEZA : BOOL ;
  A0 : BOOL ;
  A1 : BOOL ;
  B0 : BOOL ;
  B1 : BOOL ;
  C0 : BOOL ;
  C1 : BOOL ;
  C2 : BOOL ;
  D0 : BOOL ;
  D1 : BOOL ;
END_VAR
VAR_OUTPUT
  Y1 : BOOL ;
  Y2 : BOOL ;
  Y3 : BOOL ;
  Y4 : BOOL ;
  Y5 : BOOL ;
  Y6 : BOOL ;
  Y7 : BOOL ;
  Y8 : BOOL ;
END_VAR
VAR
  KA : BOOL ;
  KB : BOOL ;
  K0 : BOOL ;
  K1 : BOOL ;
  K2 : BOOL ;
  K3 : BOOL ;
END_VAR
BEGIN
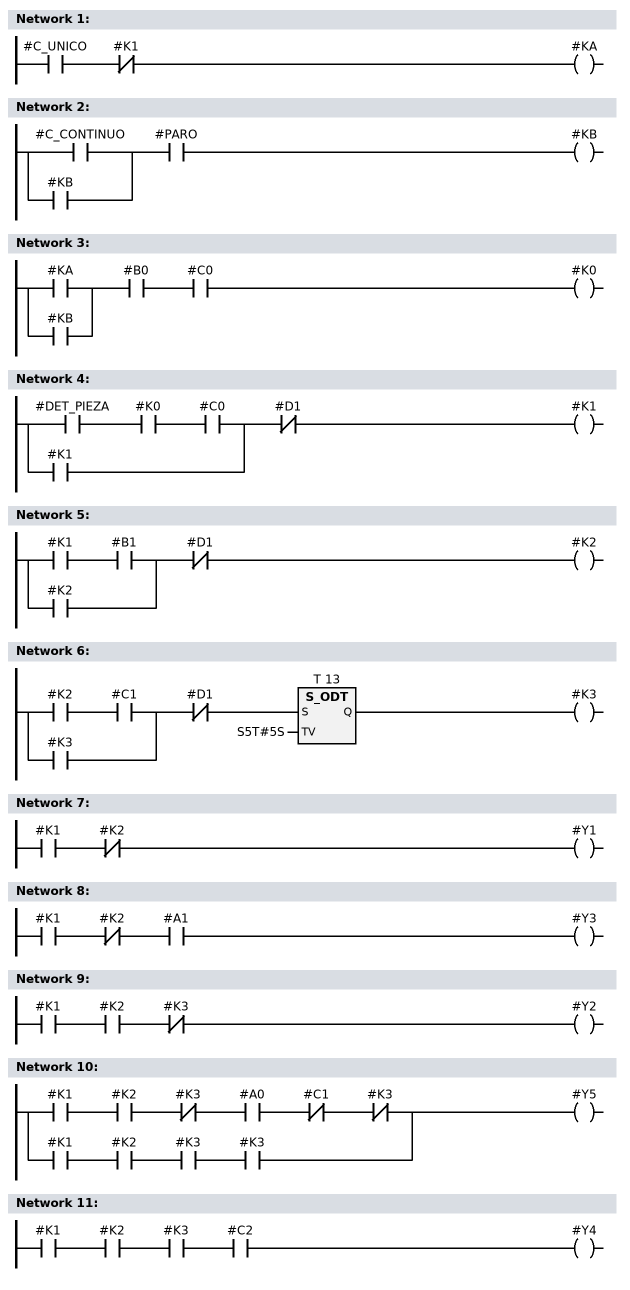
NETWORK
TITLE =
      A     #C_UNICO;
      AN    #K1;
      =     #KA;
NETWORK
TITLE =
      A(;
      O     #C_CONTINUO;
      O     #KB;
      );
      A     #PARO;
      =     #KB;
NETWORK
TITLE =
      A(;
      O     #KA;
      O     #KB;
      );
      A     #B0;
      A     #C0;
      =     #K0;
NETWORK
TITLE =
      A(;
      A     #DET_PIEZA;
      A     #K0;
      A     #C0;
      O     #K1;
      );
      AN    #D1;
      =     #K1;
NETWORK
TITLE =
      A(;
      A     #K1;
      A     #B1;
      O     #K2;
      );
      AN    #D1;
      =     #K2;
NETWORK
TITLE =
      A(;
      A     #K2;
      A     #C1;
      O     #K3;
      );
      AN    #D1;
      L     S5T#5S;
      SD    T 13;
      NOP   0;
      NOP   0;
      NOP   0;
      A     T 13;
      =     #K3;
NETWORK
TITLE =
      A     #K1;
      AN    #K2;
      =     #Y1;
NETWORK
TITLE =
      A     #K1;
      AN    #K2;
      A     #A1;
      =     #Y3;
NETWORK
TITLE =
      A     #K1;
      A     #K2;
      AN    #K3;
      =     #Y2;
NETWORK
TITLE =
      A     #K1;
      A     #K2;
      AN    #K3;
      A     #A0;
      AN    #C1;
      AN    #K3;
      O;
      A     #K1;
      A     #K2;
      A     #K3;
      A     #K3;
      =     #Y5;
NETWORK
TITLE =
      A     #K1;
      A     #K2;
      A     #K3;
      A     #C2;
      =     #Y4;
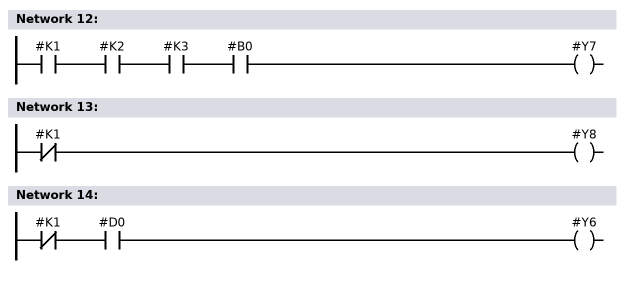
NETWORK
TITLE =
      A     #K1;
      A     #K2;
      A     #K3;
      A     #B0;
      =     #Y7;
NETWORK
TITLE =
      AN    #K1;
      =     #Y8;
NETWORK
TITLE =
      AN    #K1;
      A     #D0;
      =     #Y6;
END_FUNCTION_BLOCK

FUNCTION_BLOCK "Ejercicio 6-1"	// FB 12
VERSION : 0.1
VAR_INPUT
  C_UNICO : BOOL ;
  A0 : BOOL ;
  A1 : BOOL ;
  B0 : BOOL ;
  B1 : BOOL ;
END_VAR
VAR_OUTPUT
  Y1 : BOOL ;
  Y2 : BOOL ;
  Y3 : BOOL ;
  Y4 : BOOL ;
END_VAR
VAR
  KA : BOOL ;
  K0 : BOOL ;
  K1 : BOOL ;
  K2 : BOOL ;
  K3 : BOOL ;
  K4 : BOOL ;
END_VAR
BEGIN
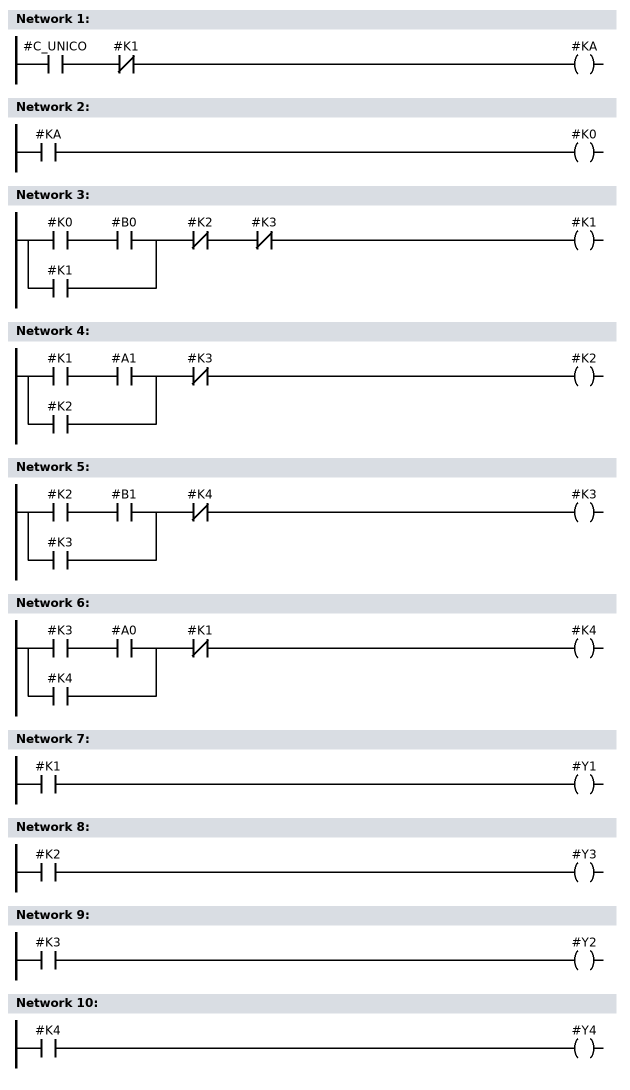
NETWORK
TITLE =
      A     #C_UNICO;
      AN    #K1;
      =     #KA;
NETWORK
TITLE =
      A     #KA;
      =     #K0;
NETWORK
TITLE =
      A(;
      A     #K0;
      A     #B0;
      O     #K1;
      );
      AN    #K2;
      AN    #K3;
      =     #K1;
NETWORK
TITLE =
      A(;
      A     #K1;
      A     #A1;
      O     #K2;
      );
      AN    #K3;
      =     #K2;
NETWORK
TITLE =
      A(;
      A     #K2;
      A     #B1;
      O     #K3;
      );
      AN    #K4;
      =     #K3;
NETWORK
TITLE =
      A(;
      A     #K3;
      A     #A0;
      O     #K4;
      );
      AN    #K1;
      =     #K4;
NETWORK
TITLE =
      A     #K1;
      =     #Y1;
NETWORK
TITLE =
      A     #K2;
      =     #Y3;
NETWORK
TITLE =
      A     #K3;
      =     #Y2;
NETWORK
TITLE =
      A     #K4;
      =     #Y4;
END_FUNCTION_BLOCK

FUNCTION_BLOCK "Ejercicio 6-2"	// FB 13
VERSION : 0.1
VAR_INPUT
  C_UNICO : BOOL ;
  A0 : BOOL ;
  A1 : BOOL ;
  B0 : BOOL ;
  B1 : BOOL ;
END_VAR
VAR_OUTPUT
  Y1 : BOOL ;
  Y2 : BOOL ;
  Y3 : BOOL ;
  Y4 : BOOL ;
END_VAR
VAR
  KA : BOOL ;
  K0 : BOOL ;
  K1 : BOOL ;
  K2 : BOOL ;
  K3 : BOOL ;
  K4 : BOOL ;
  K5 : BOOL ;
END_VAR
BEGIN
